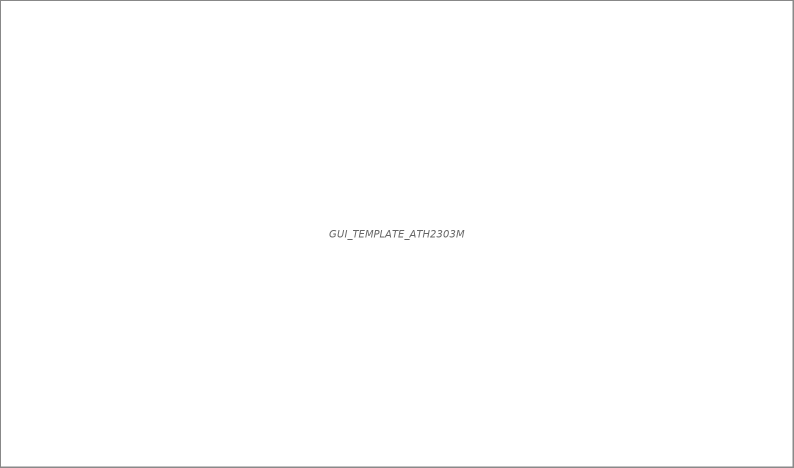
VISUALIZATION GUI_ATH2303M_EVAC_LAB  // 794x468
    Frame (0,0 794x468)
        shows GUI_TEMPLATE_ATH2303M(m_Instance := MAIN.evac_lab.tp, m_bEnable := MAIN.evac_lab.ctrl.bEnable_TP)
END_VISUALIZATION

(* stored: Version 1.1.0.1, ProductVersion 3.1.4024.9
   Visu GUI_ATH2303M_EVAC_LAB: Id {a9efa6b0-054d-400b-af67-959ea6fb63fa} *)
